FUNCTION A_BYTE : ST_Arg
VAR_INPUT
	nNumber	: REFERENCE TO BYTE;
END_VAR

IF __ISVALIDREF(nNumber) THEN
	A_BYTE.eType := E_ArgType.ByteArg;
	A_BYTE.pData := ADR(nNumber);
	A_BYTE.nSize := SIZEOF(BYTE);
END_IF

END_FUNCTION

(* stored: Version 1.1.0.1, ProductVersion 3.1.4024.15
   POU A_BYTE: Id {679824f7-b8ad-45c8-b620-fa2d53625031}, SpecialFunc None *)
